Staubli VAL3: SplitTrsf.pgx

public program SplitTrsf(string x_sSLine, string x_sTitle, trsf& x_trTrsf, bool& x_bRes)
  local string l_sChar[2]
  local num l_nData[25]
begin
  x_bRes=false

  if x_sSLine==""
    return
  endIf

  x_sSLine=right(x_sSLine,len(x_sSLine)-len(x_sTitle))

  //解析每一行
  l_sChar[0]=","
  l_sChar[1]=","

  call SplitNumS(x_sSLine,l_nData,l_sChar,x_bRes)

  if !x_bRes
    return
  endIf

  x_trTrsf.x=l_nData[0]
  x_trTrsf.y=l_nData[1]
  x_trTrsf.z=l_nData[2]
  x_trTrsf.rx=l_nData[3]
  x_trTrsf.ry=l_nData[4]
  x_trTrsf.rz=l_nData[5]




end
